ABB RobotStudio station: Practica3Avanzada_jescarcar5.rspag

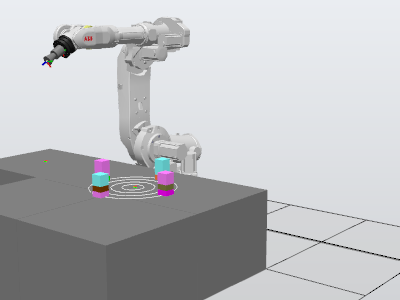
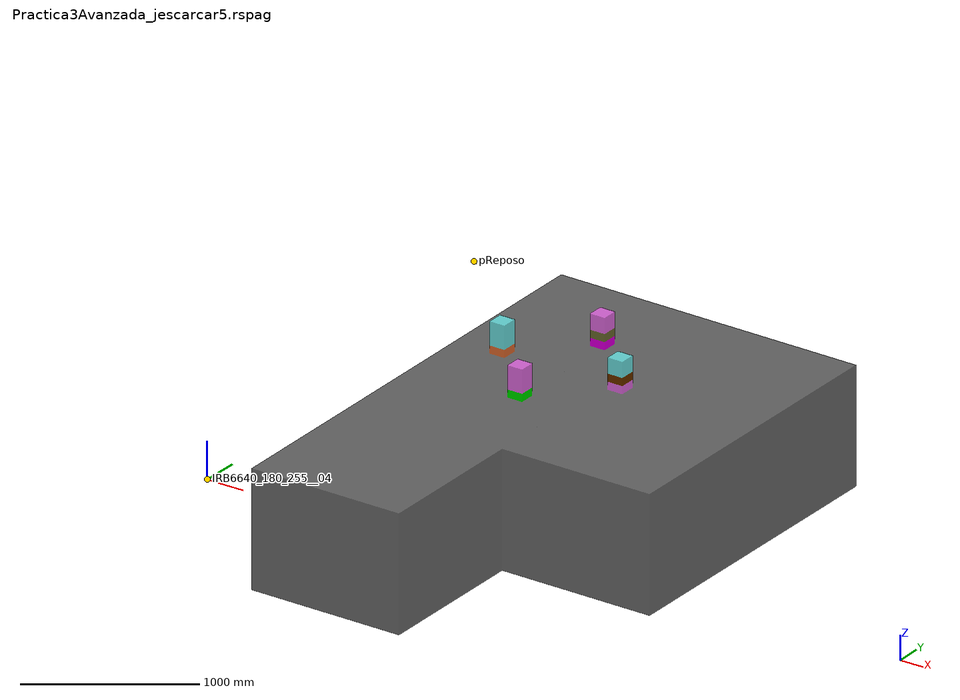
[picture v1: parts stored in the station drawn from their meshes, with robot base, taught points and paths (robot models come from the ABB library and are not in the file)]
--- station ---
Station Practica3Avanzada_EstacionDePartida (saved by RobotStudio 24.1.10713.1)
Controller Sistema6
  mechanical unit ROB_1: IRB6640_180_255__04, 6 joints, base frame (0, 0, 0) mm
Layout (positions relative to the parent item):
  - Ventosa [mechanism] at (1635.71, 0, 1955) mm, rotated rx 180 ry 60 rz 180 deg
      TCP Ventosa at (0, 0, 200) mm
      links: PiezaVentosa
  - IRB6640_180_255__04 [mechanism, from %ABB.RobotStudio.Models.IRB6640%\IRB6640_180_255_G_04.rslib] at (0, 0, 0) mm; joint values [0, 0, 0, 0, 0.5236, 0] (rad or m)
  - MesaTrabajoParte1 [part], size 1000 x 1000 x 750 mm
  - MesaTrabajoParte0 [part], size 1000 x 1000 x 750 mm
  - CI_VentosaVacuostato [smart component]
      signals: DI ActivaVentosa, DO Vacuostato
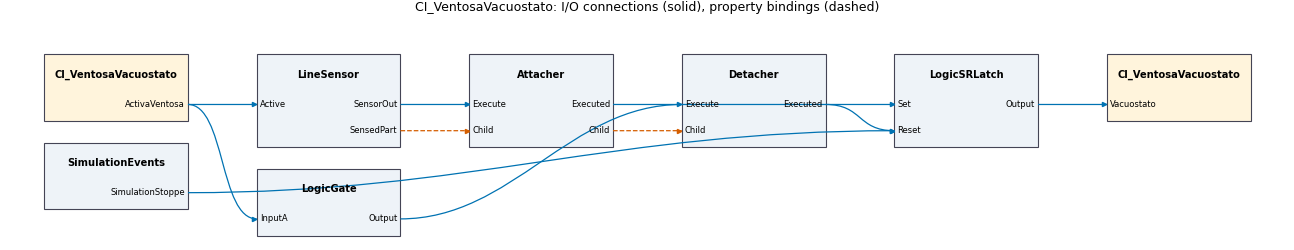
      connections:
        CI_VentosaVacuostato.ActivaVentosa -> LineSensor.Active
        LineSensor.SensorOut -> Attacher.Execute
        Attacher.Executed -> LogicSRLatch.Set
        LogicSRLatch.Output -> CI_VentosaVacuostato.Vacuostato
        Detacher.Executed -> LogicSRLatch.Reset
        SimulationEvents.SimulationStopped -> LogicSRLatch.Reset
        CI_VentosaVacuostato.ActivaVentosa -> LogicGate.InputA
        LogicGate.Output -> Detacher.Execute
        LineSensor.SensedPart => Attacher.Child
        Attacher.Child => Detacher.Child
    - LineSensor [smart component, from Components\LineSensor.rslib] at (1808.91, 0, 1855) mm, rotated rx 180 ry 60 rz 180 deg
        properties: Start=[0 0 -0.002]; End=[0 0 0.02]; Radius=0.002; SensedPart=Pieza1; SensedPoint=[1.69999987792969 0.6 0.95]; Length=0.022; Tag=(none)
      - _sensorPart_ [part], size 4 x 4 x 22 mm
    - SimulationEvents [smart component, from Components\SimulationEvents.rslib]
    - LogicSRLatch [smart component, from Components\LogicSRLatch.rslib]
    - Attacher [smart component, from Components\Attacher.rslib]
        properties: Parent=Ventosa; Flange=0; Child=Pieza1; Mount=false; Offset=[0 0 0]; Orientation=[0 0 0]
    - Detacher [smart component, from Components\Detacher.rslib]
        properties: Child=Pieza1; KeepPosition=true
    - LogicGate [smart component, from Components\LogicGate.rslib]
        properties: Operator=NOT; Delay=0.1
  - MesaTrabajoParte2 [part] at (0, 1000, 0) mm, size 1000 x 1000 x 750 mm
  - MesaTrabajoParte3 [part] at (1000, 0, 0) mm, size 1000 x 1000 x 750 mm
  - MesaTrabajoParte4 [part] at (1000, 1000, 0) mm, size 1000 x 1000 x 750 mm
  - Pieza1 [part] at (200, 1100, 150) mm, size 100 x 100 x 50 mm
  - Pieza2 [part] at (-200, 1500, 100) mm, size 100 x 100 x 50 mm
  - Pieza3 [part] at (200, 1900, 50) mm, size 100 x 100 x 50 mm
  - Pieza4 [part] at (600, 1500, 0) mm, size 100 x 100 x 50 mm
  - Pieza5 [part] at (200, 1100, -100) mm, size 100 x 100 x 50 mm
  - CircunferenciaR200 [part], size 400 x 400 x 0 mm
  - CircunferenciaR100 [part], size 200 x 198.9 x 0 mm
  - CircunferenciaR300 [part], size 599 x 599.5 x 0 mm
  - CircunferenciaR400 [part], size 799 x 799.5 x 0 mm
  - Pieza6 [part] at (-200, 1500, -150) mm, size 100 x 100 x 50 mm
  - Pieza7 [part] at (200, 1900, -200) mm, size 100 x 100 x 50 mm
  - Pieza8 [part] at (600, 1500, -250) mm, size 100 x 100 x 50 mm
  - Pieza9 [part] at (200, 1100, -350) mm, size 100 x 100 x 50 mm
  - Pieza10 [part] at (-200, 1500, -400) mm, size 100 x 100 x 50 mm
  - Pieza10_2 [part] at (200, 1900, -400) mm, size 100 x 100 x 50 mm
  - Pieza10_5 [part] at (600, 1500, -400) mm, size 100 x 100 x 50 mm
  - Pieza10_6 [part] at (200, 1100, -450) mm, size 100 x 100 x 50 mm
  - Pieza10_7 [part] at (-200, 1500, -450) mm, size 100 x 100 x 50 mm
  - Pieza10_8 [part] at (200, 1900, -450) mm, size 100 x 100 x 50 mm
  - Pieza10_9 [part] at (600, 1500, -450) mm, size 100 x 100 x 50 mm
Attachment: Ventosa is attached to IRB6640_180_255__04 / Link6
Attachment: LineSensor is attached to Ventosa / PiezaVentosa
Station logic (signal -> signal, property => property):
  CI_VentosaVacuostato.Vacuostato -> Sistema6.ED_PiezaCogida
  Sistema6.SD_ActivaVentosa -> CI_VentosaVacuostato.ActivaVentosa

--- Backups/Sistema6/RAPID/TASK1/PROGMOD/CalibData.mod ---
MODULE CalibData
	PERS tooldata Ventosa:=[TRUE,[[0,0,200],[1,0,0,0]],[1,[0,0,125],[1,0,0,0],0.002,0.002,0.0013]];
ENDMODULE

--- Backups/Sistema6/RAPID/TASK1/PROGMOD/Module1.mod ---
MODULE Module1
    CONST robtarget pBaseOrigen:=[[1500,-500,750],[0,0,1,0],[0,0,0,0],[9E+09,9E+09,9E+09,9E+09,9E+09,9E+09]];
    CONST robtarget pCentroDestino:=[[1700,1000,750],[0,0,1,0],[0,0,0,0],[9E+09,9E+09,9E+09,9E+09,9E+09,9E+09]];
    CONST robtarget pReposo:=[[1808.910161514,0,1855],[0.5,0,0.866025404,0],[0,0,0,0],[9E+09,9E+09,9E+09,9E+09,9E+09,9E+09]];
    VAR num altoPieza := 50;
    var num nPiezasTorreOrigen := 16;
    CONST num nTorresDestino := 4;
    var num radioCircunf := 400;
    VAR robtarget posicionesDestino{nTorresDestino};
    PROC MAIN()
        SetDO SD_ActivaVentosa, 0;
        MoveJ pReposo, v1000,z50,Ventosa;
        TrasladaTorre pBaseOrigen,pCentroDestino,pReposo,altoPieza,nPiezasTorreOrigen,nTorresDestino,radioCircunf;
        MoveJ pReposo, v1000,z50,Ventosa;
        SetDO SD_ActivaVentosa, 0;
    ENDPROC
    PROC TrasladaTorre( robtarget pBaseOrigen,robtarget pCentroDestino,robtarget pReposo,num altoPieza,num nPiezasTorreOrigen,num nTorresDestino,num radioCircunf)

        VAR num x;
        VAR robtarget pOrigen;
        VAR robtarget pDestino;

       CalcularPosicionesDestino radioCircunf,nTorresDestino, pCentroDestino;
       FOR  i FROM 1 TO nPiezasTorreOrigen DO
            x := ((i-1)MOD nTorresDestino) +1;
            pOrigen:= pBaseOrigen;
            pOrigen.trans.z := pBaseOrigen.trans.z +((nPiezasTorreOrigen-i+1)*altoPieza);
            pDestino:= posicionesDestino{x};
            pDestino.trans.z := pDestino.trans.z +altoPieza;
            muevePieza pOrigen,pDestino;
            posicionesDestino{x}:= pDestino;
       ENDFOR
    ENDPROC

        PROC CalcularPosicionesDestino(num radioCircunf,num nTorresDestino,robtarget pCentroDestino)
        VAR num angulo;
         VAR robtarget pAux;

        FOR i FROM 1 TO nTorresDestino DO
            pAux:= pCentroDestino;
            angulo := (360 / nTorresDestino) * (i - 1);
            pAux.trans.x := pCentroDestino.trans.x + radioCircunf * Cos(angulo);
            pAux.trans.y := pCentroDestino.trans.y + radioCircunf * Sin(angulo);
            pAux.trans.z:= pCentroDestino.trans.z;
            posicionesDestino{i} := pAux;
        ENDFOR
    ENDPROC

        PROC muevePieza(robtarget pOrigen,robTarget pDestino)
            VAR robtarget pOrigenAprox;
            VAR robtarget pDestinoAprox;
            VAR num alturaAprox:= 150;
            pOrigenAprox := pOrigen;
             pDestinoAprox := pDestino;
            pOrigenAprox.trans.z := pOrigen.trans.z + alturaAprox;
            pDestinoAprox.trans.z := pDestino.trans.z + alturaAprox;
            MoveJ pOrigenAprox,v2000,z100,Ventosa\WObj:=wobj0;
            MoveL pOrigen,v300,fine,Ventosa\WObj:=wobj0;
            SetDO SD_ActivaVentosa, 1;! se puede combinar con mode LDO
            WaitDI ED_PiezaCogida, 1;
            MoveL pOrigenAprox,v300,z0,Ventosa\WObj:=wobj0;
            MoveJ pDestinoAprox,v2000,z100,Ventosa\WObj:=wobj0;
            MoveL pDestino,v300,fine,Ventosa\WObj:=wobj0;
            SetDO SD_ActivaVentosa, 0;
            WaitDI ED_PiezaCogida, 0;
            MoveL pDestinoAprox,v300,fine,Ventosa\WObj:=wobj0;
    ENDPROC
ENDMODULE

--- Backups/Sistema6/RAPID/TASK1/SYSMOD/LINKEDM.sys ---
%%%
  VERSION:1
  LANGUAGE:ENGLISH
%%%

MODULE LINKEDM (SYSMODULE)

! FOLLOWER
!     Name of electronically linked follower axis used by operator at teach pendent.
      PERS string l_f_axis_name{5}       :=  ["",  "", "", "", ""];

!     Name of the mechanical unit for follower axis.
      PERS string l_f_mecunt_n{5}  :=  ["", "", "", "", ""];

!     Linked follower axis number in the mechanical unit (first axis in mech. unit is number 1).
      PERS num l_f_axis_no{5}      :=  [0,          0,   0,  0,  0];

! MASTER
!     Name of the mechanical unit for linked master axis.
      PERS string l_m_mecunt_n{5} :=  ["", "", "", "", ""];

!     Linked master axis number in the mechanical unit (first axis in mech. unit is number 1).
!     See axis number table in documentation for different master mechanical units.
      PERS num l_m_axis_no{5}     :=  [0,  0,  0,  0,  0];

! POSITION OFFSET
!     The increase of the allowed offset position between the master and follower
!     positions, used when starting AUTO mode. As soon as the offset is decreased
!     the old configurated parameter is used.
!     Example: 3 => the configurated value of allowed offset is increased 3 times.
      PERS num offset_ratio{5}       :=  [10,  10,   10,  10,  10];

! SPEED RATIO
!     Speed_ratio used in AUTO and JOG modes [ very_slow   slow    normal    fast]
!     Value 1 = max allowed manual speed.
      CONST num speed_ratio {20}      := [0.01, 0.01, 0.01, 0.01, 0.01,
                                          0.05, 0.05, 0.05, 0.05, 0.05,
                                          0.20, 0.20, 0.20, 0.20, 0.20,
                                          1.00, 1.00, 1.00, 1.00, 1.00];

! STEP SIZE
!     Displacement position used in JOG mode for each activation of positive or
!     negative movement.                  [very_short    short   normal   long]
!     Unit degees or meter.
      CONST num displacement {20}     := [0.001, 0.001, 0.001, 0.001, 0.001,
                                          0.005, 0.005, 0.005, 0.005, 0.005,
                                          0.020, 0.020, 0.020, 0.020, 0.020,
                                          0.100, 0.100, 0.100, 0.100, 0.100];


!-------------------------------------------------------------
 PROC Linked_m ()
      Linked_m_exe ;
 ENDPROC
ENDMODULE

--- Backups/Sistema6/SYSPAR/EIO.cfg ---
EIO:CFG_1.0:6:1::
#
INDUSTRIAL_NETWORK:

      -Name "DeviceNet" -Label "DeviceNet Master/Slave Network" -Address "2"
#
DEVICENET_DEVICE:

      -Name "MiDeviceNet" -Label "MiDeviceNet"
#
DEVICENET_INTERNAL_DEVICE:

      -Name "DN_Internal_Device" -VendorName "ABB Robotics"\
      -ProductName "DeviceNet Internal Slave Device"
#
EIO_SIGNAL:

      -Name "ED_PiezaCogida" -SignalType "DI" -Device "MiDeviceNet"\
      -Label "ED_PiezaCogida" -DeviceMap "0" -Access "All"

      -Name "SD_ActivaVentosa" -SignalType "DO" -Device "MiDeviceNet"\
      -Label "SD_ActivaVentosa" -DeviceMap "0" -Access "All"
